(* PLC project FidelityFixture, greenforge-labs codescribe-fixture 1 *)
(* stored: creationDateTime 2020-01-01T00:00:00 *)

PROGRAM FBD_FIDELITY
  VAR_INPUT
    xIn : BOOL;
  END_VAR

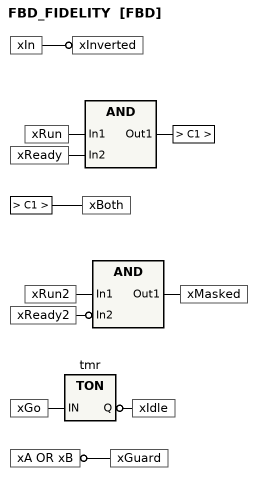
(* FBD diagram, written out as Structured Text *)
xInverted := NOT xIn;
xBoth := xRun AND xReady;
xMasked := xRun2 AND NOT xReady2;
tmr(IN := xGo, Q => xIdle);
xGuard := NOT (xA OR xB);
END_PROGRAM
